FUNCTION_BLOCK FB_State_IOs
VAR_INPUT
END_VAR
VAR_OUTPUT
END_VAR
VAR
	out_sts AT %Q* : BYTE;
END_VAR

END_FUNCTION_BLOCK

(* stored: Version 1.1.0.1, ProductVersion 3.1.4024.12
   POU FB_State_IOs: Id {743b422d-0aca-40cd-9426-4749e414f45b}, SpecialFunc None *)
